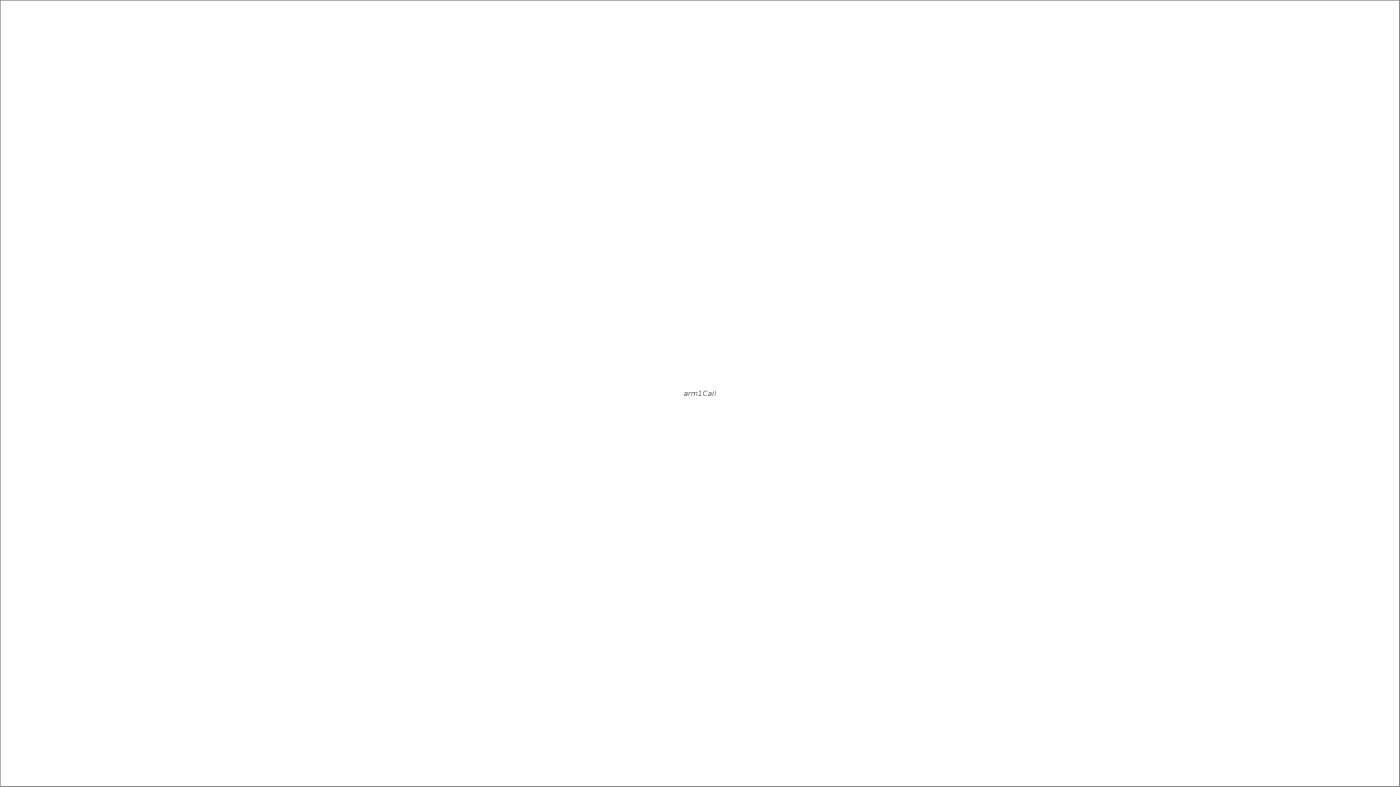
VISUALIZATION robotCail  // 1920x1080
    TabControl (0,0 1920x1080)
        shows arm1Cail()
        shows arm2Cail()
        shows arm3Cail()
        shows arm4Cail()
        shows carCail()
END_VISUALIZATION

(* stored: Version 1.1.0.1, ProductVersion 3.1.4024.11
   Visu robotCail: Id {2258b39a-017c-4eed-8f75-7343650db6b1} *)
